(* CoDeSys 2.3.9.62 project: Tema1 Ejemplo2-Deposito v0.pro *)

(* Global variable list: Global_Variables *)
VAR_GLOBAL
  N1:BOOL;
  N2:BOOL;
  Bomba:BOOL;
  Bomba1:BOOL;
  M :BOOL;
END_VAR

(* POU PLC_PRG, ST *)
PROGRAM PLC_PRG
VAR
  posy:INT;

	Desague: BOOL;
END_VAR
Control();


IF Bomba=TRUE THEN
IF posy>-187 THEN
  posy:=posy-1;
END_IF
END_IF

IF Bomba=FALSE THEN
IF posy<52 THEN
  posy:=posy+1;
END_IF
END_IF

IF Bomba1=TRUE THEN
IF posy>-187 THEN
  posy:=posy-1;
END_IF
END_IF


IF Desague=1 THEN
IF posy<48 THEN
posy:=posy+4;
END_IF
END_IF

IF posy<-121 THEN
  N2:=TRUE;
ELSE
  N2:=FALSE;
END_IF

IF posy<-166 THEN
  N1:=TRUE;
ELSE
  N1:=FALSE;
END_IF
END_PROGRAM

(* POU Control, LD *)
PROGRAM Control
VAR
    KM1:BOOL;
	B: BOOL;
	N: BOOL;
END_VAR
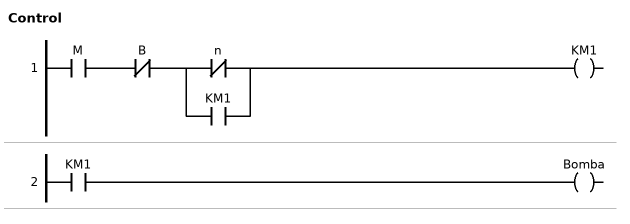
_LD_ (* Ladder Diagram *)
NETWORK 1
	[M] - [/B] - { [/n] | [KM1] } --- (KM1)
NETWORK 2
	[KM1] --- (Bomba)
_END_LD_
(* the same logic as Structured Text *)
(* Network 1 *)
KM1 := M AND NOT B AND (NOT n OR KM1);
(* Network 2 *)
Bomba := KM1;
END_PROGRAM

(* Visualisation Deposito
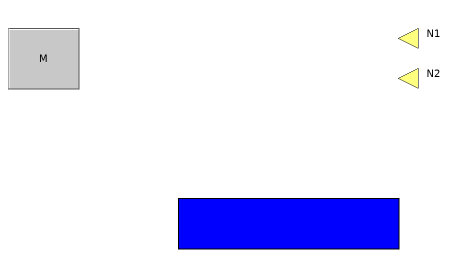
button at (50,80)-(121,141): text "M"; toggles M
polygon at (440,80)-(460,100): alarm colour if .N1; toggles .B
polygon at (440,120)-(460,140): alarm colour if .N2; toggles .A
rectangle at (460,70)-(491,101): text "N1"
rectangle at (460,110)-(491,141): text "N2"
rectangle at (220,250)-(441,301): top PLC_PRG.posy
1 more shapes without text or variables
1 elements of other kinds (tables, trends, ...) not read
*)
